FUNCTION_BLOCK FB_ZAE
VAR_INPUT

END_VAR
VAR_OUTPUT

END_VAR
VAR
	{attribute 'OPC.UA.DA' := '1'}BHKW_321_SZ_Zustand			: ST_SZ_Zustand;
	{attribute 'OPC.UA.DA' := '1'}BHKW_322_SZ_Zustand			: ST_SZ_Zustand;
	{attribute 'OPC.UA.DA' := '1'}Gebaeude_SZ_Zustand			: ST_SZ_Zustand;
	{attribute 'OPC.UA.DA' := '1'}Buerotrakt_SZ_Zustand		: ST_SZ_Zustand;	
	{attribute 'OPC.UA.DA' := '1'}Halle_TGA_SZ_Zustand		: ST_SZ_Zustand;	
	{attribute 'OPC.UA.DA' := '1'}Halle_Licht_SZ_Zustand		: ST_SZ_Zustand;
	{attribute 'OPC.UA.DA' := '1'}BHKW_1_GZ_Zustand			: ST_GZ_Zustand;	
	{attribute 'OPC.UA.DA' := '1'}BHKW_2_GZ_Zustand			: ST_GZ_Zustand;	
	{attribute 'OPC.UA.DA' := '1'}DLK_Gaszaehler_Zustand		: ST_GZ_DLK_Zustand;
	{attribute 'OPC.UA.DA' := '1'}Stromzaehler_NSHV_Zustand	: ST_NSHV_Zustand;		
	{attribute 'OPC.UA.DA' := '1'}WP_946_WZ_4371_Zustand		: ST_WZ_Zustand;	
	{attribute 'OPC.UA.DA' := '1'}WP_946_WZ_4372_Zustand		: ST_WZ_Zustand;	
                                                                                    
	{attribute 'OPC.UA.DA' := '1'}Brennwerttherme_WZ_Zustand	: ST_WZ_Zustand;	
	{attribute 'OPC.UA.DA' := '1'}BHKW_1_WZ_Zustand			: ST_WZ_Zustand;		
	{attribute 'OPC.UA.DA' := '1'}BHKW_2_WZ_Zustand			: ST_WZ_Zustand;		
	{attribute 'OPC.UA.DA' := '1'}Druckluftkompressor_WZ_Zustand			: ST_WZ_Zustand;
	{attribute 'OPC.UA.DA' := '1'}PWT_1_WZ_Zustand			: ST_WZ_Zustand;				
	{attribute 'OPC.UA.DA' := '1'}Ofenkuehlung_WZ_Zustand		: ST_WZ_Zustand;			
	{attribute 'OPC.UA.DA' := '1'}Abgasfackel_WZ_Zustand		: ST_WZ_Zustand;			
                                                                                    			
	Stromzaehler_BHKW_321		: FB_Stromzaehler_BHKW;
	Stromzaehler_Gebaeude		: FB_Stromzaehler_Gebaeude;
	Stromzaehler_Buerotrakt		: FB_Stromzaehler;
	Stromzaehler_BHKW_322		: FB_Stromzaehler_BHKW;
	Stromzaehler_Halle_TGA		: FB_Stromzaehler;
	Stromzaehler_Halle_Licht	: FB_Stromzaehler;
	Gaszaehler_BHKW_1			: FB_Gaszaehler;
	Gaszaehler_BHKW_2			: FB_Gaszaehler;
	Gaszaehler_DLK				: FB_GZ_DLK;
	Stromzaehler_NSHV_Modbus	: FB_Stromzaehler_NSHV_Modbus;

	Waermezaehler_4371_WP_946	: FB_Waermezaehler_WP;
	Waermezaehler_4372_WP_946	: FB_Waermezaehler_WP;

	Waermezaehler_331_Brennwerttherme	: FB_Waermezaehler_MollineC3;
	Waermezaehler_321_BHKW_1			: FB_Waermezaehler_MollineC3;
	Waermezaehler_322_BHKW_2			: FB_Waermezaehler_MollineC3;
	Waermezaehler_251_Druckluftkompressor	: FB_Waermezaehler_MollineC3;
	Waermezaehler_215_PWT_1				: FB_Waermezaehler_MollineC3;
	Waermezaehler_261_Ofenkuehlung		: FB_Waermezaehler_MollineC3;
	Waermezaehler_361_Ofen_Abgasfackel	: FB_Waermezaehler_MollineC3;
END_VAR

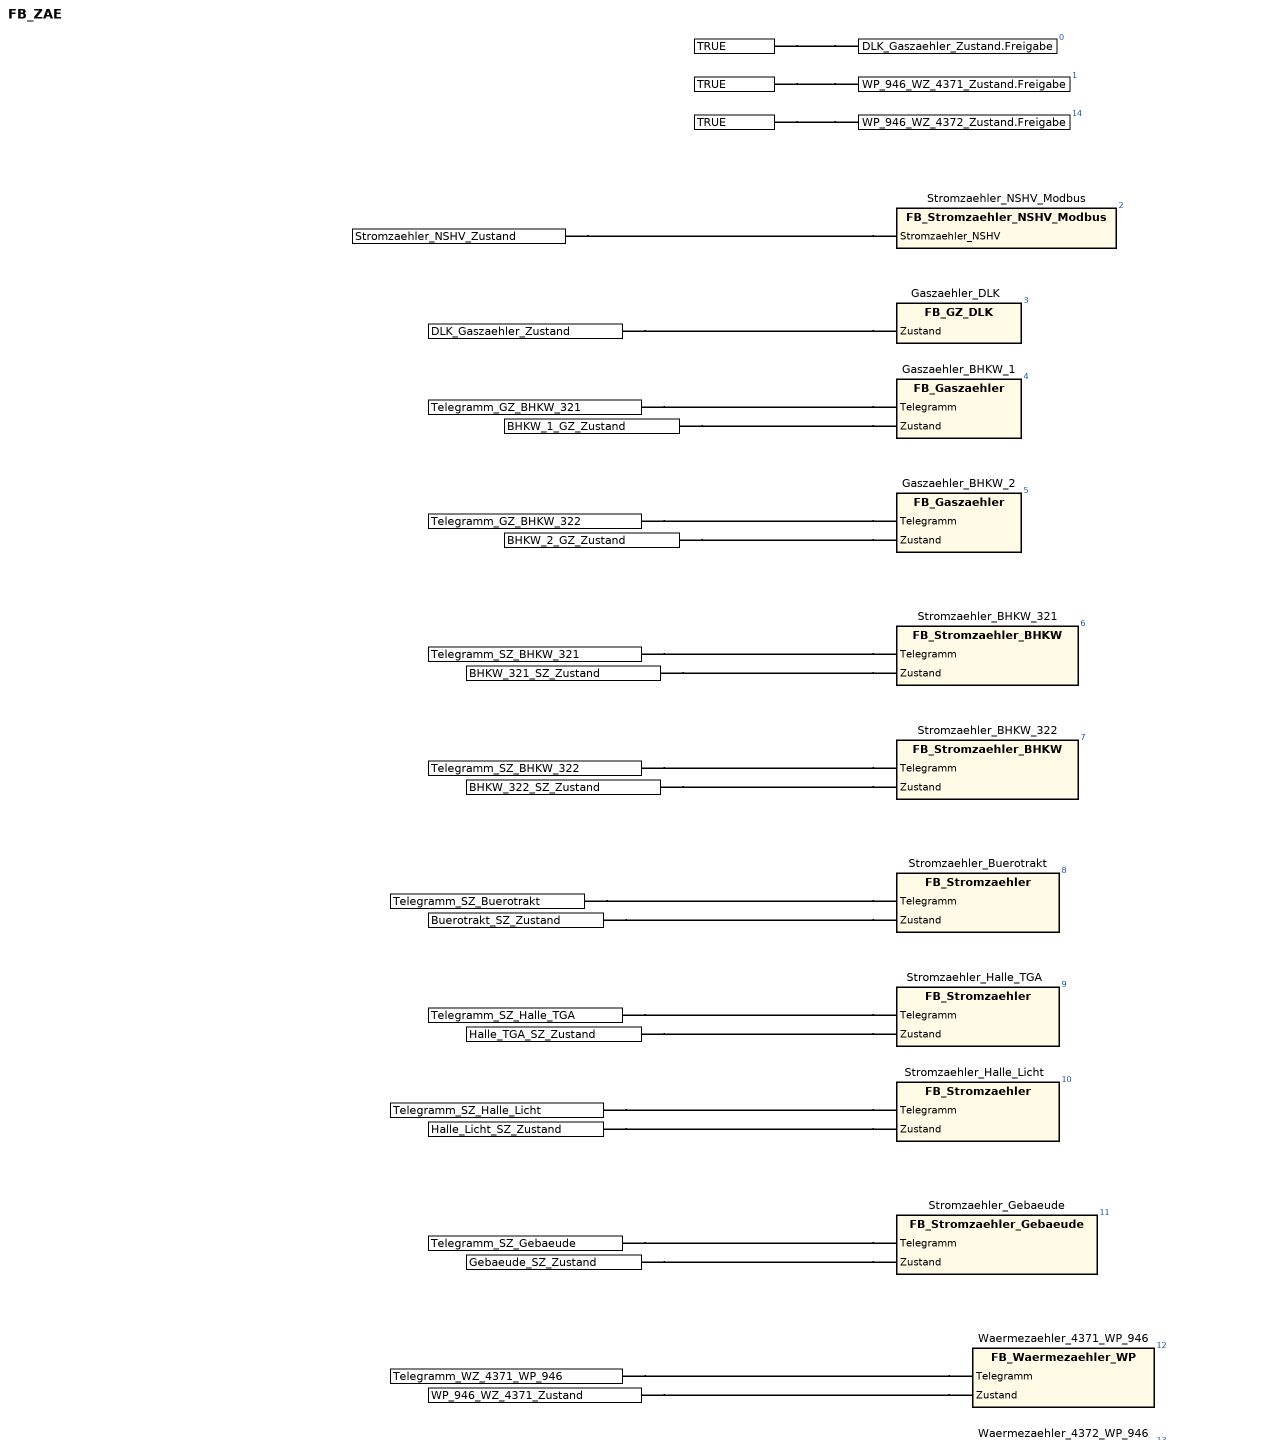
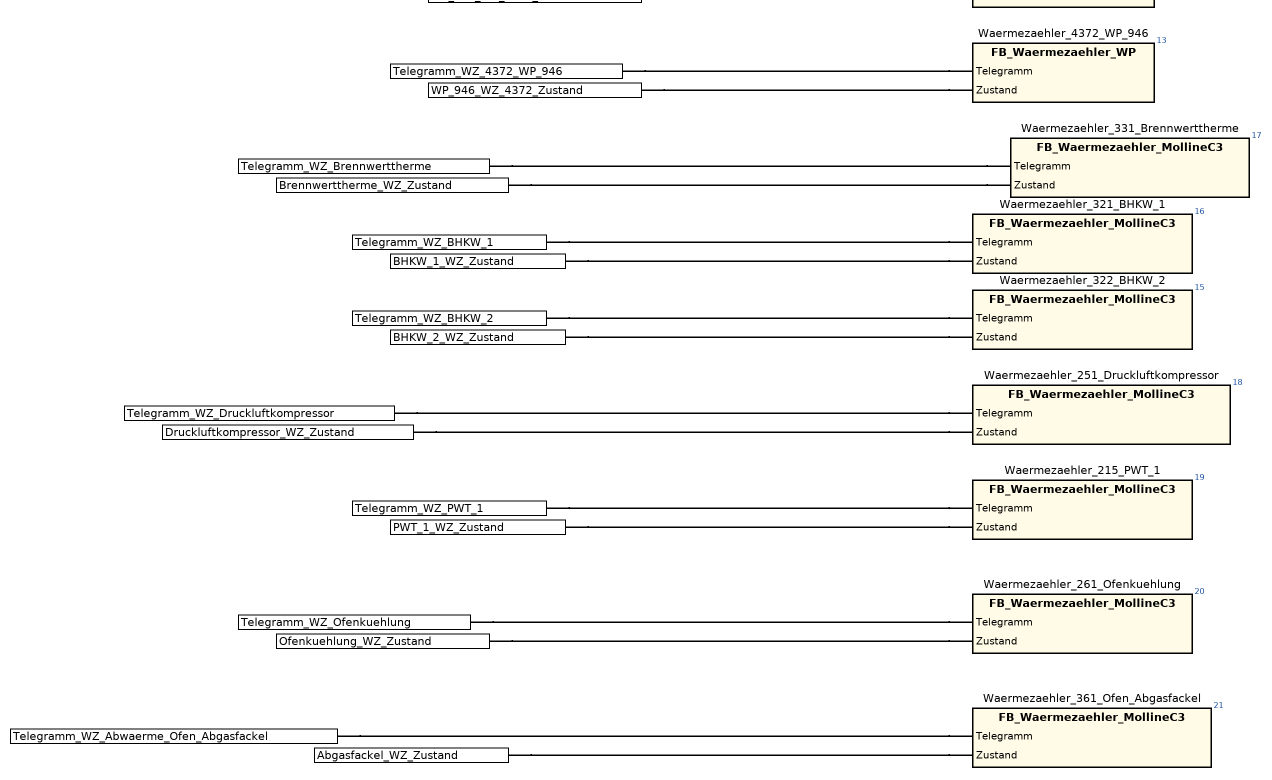
DLK_Gaszaehler_Zustand.Freigabe := TRUE;
WP_946_WZ_4371_Zustand.Freigabe := TRUE;
Stromzaehler_NSHV_Modbus(Stromzaehler_NSHV := Stromzaehler_NSHV_Zustand); // FB_Stromzaehler_NSHV_Modbus
Gaszaehler_DLK(Zustand := DLK_Gaszaehler_Zustand); // FB_GZ_DLK
Gaszaehler_BHKW_1(Telegramm := Telegramm_GZ_BHKW_321, Zustand := BHKW_1_GZ_Zustand); // FB_Gaszaehler
Gaszaehler_BHKW_2(Telegramm := Telegramm_GZ_BHKW_322, Zustand := BHKW_2_GZ_Zustand); // FB_Gaszaehler
Stromzaehler_BHKW_321(Telegramm := Telegramm_SZ_BHKW_321, Zustand := BHKW_321_SZ_Zustand); // FB_Stromzaehler_BHKW
Stromzaehler_BHKW_322(Telegramm := Telegramm_SZ_BHKW_322, Zustand := BHKW_322_SZ_Zustand); // FB_Stromzaehler_BHKW
Stromzaehler_Buerotrakt(Telegramm := Telegramm_SZ_Buerotrakt, Zustand := Buerotrakt_SZ_Zustand); // FB_Stromzaehler
Stromzaehler_Halle_TGA(Telegramm := Telegramm_SZ_Halle_TGA, Zustand := Halle_TGA_SZ_Zustand); // FB_Stromzaehler
Stromzaehler_Halle_Licht(Telegramm := Telegramm_SZ_Halle_Licht, Zustand := Halle_Licht_SZ_Zustand); // FB_Stromzaehler
Stromzaehler_Gebaeude(Telegramm := Telegramm_SZ_Gebaeude, Zustand := Gebaeude_SZ_Zustand); // FB_Stromzaehler_Gebaeude
Waermezaehler_4371_WP_946(Telegramm := Telegramm_WZ_4371_WP_946, Zustand := WP_946_WZ_4371_Zustand); // FB_Waermezaehler_WP
Waermezaehler_4372_WP_946(Telegramm := Telegramm_WZ_4372_WP_946, Zustand := WP_946_WZ_4372_Zustand); // FB_Waermezaehler_WP
WP_946_WZ_4372_Zustand.Freigabe := TRUE;
Waermezaehler_322_BHKW_2(Telegramm := Telegramm_WZ_BHKW_2, Zustand := BHKW_2_WZ_Zustand); // FB_Waermezaehler_MollineC3
Waermezaehler_321_BHKW_1(Telegramm := Telegramm_WZ_BHKW_1, Zustand := BHKW_1_WZ_Zustand); // FB_Waermezaehler_MollineC3
Waermezaehler_331_Brennwerttherme(Telegramm := Telegramm_WZ_Brennwerttherme, Zustand := Brennwerttherme_WZ_Zustand); // FB_Waermezaehler_MollineC3
Waermezaehler_251_Druckluftkompressor(Telegramm := Telegramm_WZ_Druckluftkompressor, Zustand := Druckluftkompressor_WZ_Zustand); // FB_Waermezaehler_MollineC3
Waermezaehler_215_PWT_1(Telegramm := Telegramm_WZ_PWT_1, Zustand := PWT_1_WZ_Zustand); // FB_Waermezaehler_MollineC3
Waermezaehler_261_Ofenkuehlung(Telegramm := Telegramm_WZ_Ofenkuehlung, Zustand := Ofenkuehlung_WZ_Zustand); // FB_Waermezaehler_MollineC3
Waermezaehler_361_Ofen_Abgasfackel(Telegramm := Telegramm_WZ_Abwaerme_Ofen_Abgasfackel, Zustand := Abgasfackel_WZ_Zustand); // FB_Waermezaehler_MollineC3

END_FUNCTION_BLOCK

(* stored: Version 1.1.0.1, ProductVersion 3.1.4024.9
   POU FB_ZAE: Id {198980c7-41f5-4a16-a8a4-0b5521f44eae}, SpecialFunc None *)
